(* Logix 5000 project; controller cal1615 1756-L62 rev 20.19; software revision 20.05; part 14 of 81 *)
(* tags used below, declared in another part *)
   FAULT : BOOL;   // Fault AFI
   HMI : BOOL;   // AFI HMI
   p00_lin_timer_pre_0ms : DINT;
   p00_lin_timer_pre_1s : DINT;
   p00_lin_timer_pre_disc : DINT;
   p00_lin_timer_pre_mcp : DINT;
   p00_lin_timer_pre_ms : DINT;
   p00_lin_timer_pre_ol : DINT;
   p01_dint_to_hmi : DINT[16];   // System Dint to HMI
   p01_recipe_active : recipe;   // Active Recipe
   p01r09_pb_global_reset : BOOL;   // System Modes PB: Global Fault Reset
   p02_dint_from_hmi : hmi_dint;
   p02_dint_to_hmi : hmi_dint;   // MOP HMI Iface Dint to HMI
   p02_recipe_from_hmi : recipe;   // MOP HMI Iface Recipe From HMI
   p02_recipe_to_hmi : recipe;   // MOP HMI Iface To HMI Recipe
   p02r01 : routine;   // MOP HMI Iface Main
   p02r02 : routine;   // MOP HMI Iface Misc Control
   p02r02_timer_fault : TIMER[4];   // MOP HMI Iface Misc Control Fault Delay
   p02r02_timer_logout : TIMER;
   p02r02_timer_warning : TIMER[4];   // MOP HMI Iface Misc Control Warning Delay
   p02r03 : routine;   // MOP HMI Iface Navigation
   p02r03_timer_fault : TIMER[4];   // MOP HMI Iface Navigation Fault Delay
   p02r03_timer_warning : TIMER[4];   // MOP HMI Iface Navigation Warning Delay
   p02r04 : routine;   // MOP HMI Iface Recipe
   p02r04_timer_fault : TIMER[4];   // MOP HMI Iface Recipe Fault Delay
   p02r04_timer_warning : TIMER[4];   // MOP HMI Iface Recipe Warning Delay
   p02r05 : routine;   // MOP HMI Iface Dint to HMI
   p02r05_timer_fault : TIMER[4];   // MOP HMI Iface Dint to HMI Fault Delay
   p02r05_timer_warning : TIMER[4];   // MOP HMI Iface Dint to HMI Warning Delay
   p02r07 : routine;   // MOP HMI Iface Alarms
   p11_dint_to_hmi : DINT[16];   // Zone 1 Temperature Control VFDs On
   p12_dint_to_hmi : DINT[16];   // Zone 2 Temperature Control VFDs On
   p13_dint_to_hmi : DINT[16];   // Zone 3 Temperature Control VFDs On
   p19_dint_to_hmi : DINT[16];
   p20_dint_to_hmi : DINT[16];   // Letoff Dint to HMI
   p21_dint_to_hmi : DINT[16];   // Splice Press
   p22_dint_to_hmi : DINT[16];   // Tension Stand 1 Dint to HMI
   p23_dint_to_hmi : DINT[17];   // Impreg Dint to HMI
   p24_dint_to_hmi : DINT[16];
   p25_dint_to_hmi : DINT[16];   // Tension Stand 2 Dint to HMI
   p26_dint_to_hmi : DINT[16];   // Upper Poly Letoff Dint to HMI
   p27_dint_to_hmi : DINT[16];   // Lower Poly Letoff Alarms
   p28_dint_to_hmi : DINT[16];
   p29_dint_to_hmi : DINT[16];   // Winder Dint to HMI
   p30_dint_to_hmi : DINT[16];   // Retraction System Dint to HMI
(* P01_System, continued *)

ROUTINE R32_LIN_Timer_Presets   (* ladder *)
// System
// System Timer Presets
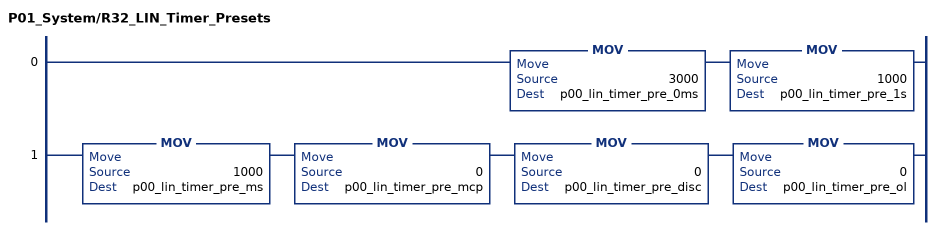
   0: MOV(3000,p00_lin_timer_pre_0ms)MOV(1000,p00_lin_timer_pre_1s);
   1: MOV(1000,p00_lin_timer_pre_ms)MOV(0,p00_lin_timer_pre_mcp)MOV(0,p00_lin_timer_pre_disc)MOV(0,p00_lin_timer_pre_ol);
END_ROUTINE
END_PROGRAM

PROGRAM P02_MOP_HMI_Iface   (* main routine R01_Main *)
VAR
   Limit_Clamp : sys_Limit_Clamp;   // Limit Clamp
END_VAR

ROUTINE R01_Main   (* ladder *)
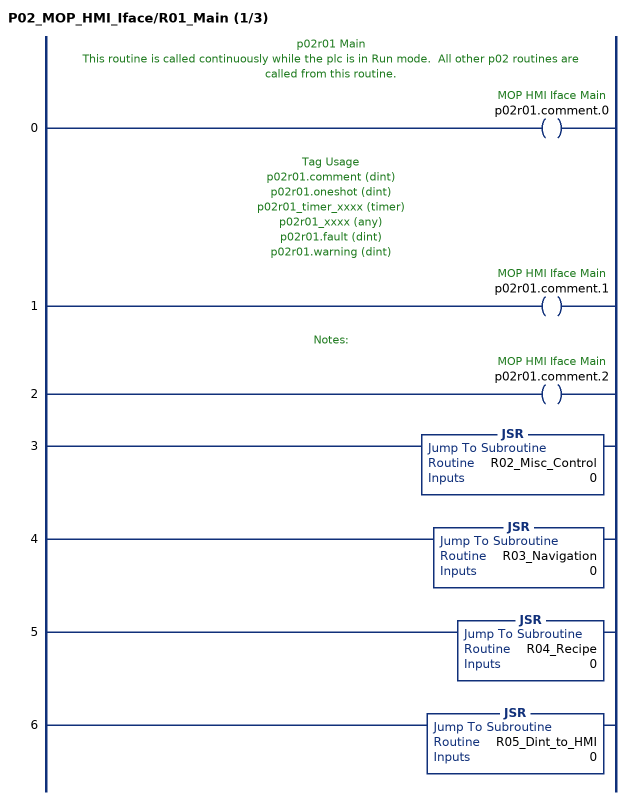
   // p02r01 Main
   // This routine is called continuously while the plc is in Run mode.  All other p02 routines are called from this routine.
   0: OTE(p02r01.comment.0);
   // Tag Usage
   // p02r01.comment (dint)
   // p02r01.oneshot (dint)
   // p02r01_timer_xxxx (timer)
   // p02r01_xxxx (any)
   // p02r01.fault (dint)
   // p02r01.warning (dint)
   1: OTE(p02r01.comment.1);
   // Notes:
   2: OTE(p02r01.comment.2);
   3: JSR(R02_Misc_Control,0);
   4: JSR(R03_Navigation,0);
   5: JSR(R04_Recipe,0);
   6: JSR(R05_Dint_to_HMI,0);
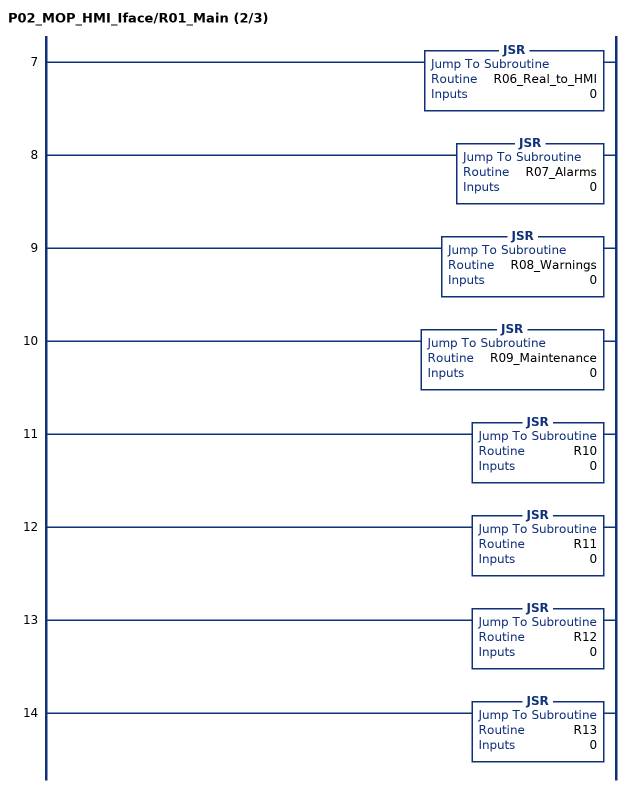
   7: JSR(R06_Real_to_HMI,0);
   8: JSR(R07_Alarms,0);
   9: JSR(R08_Warnings,0);
   10: JSR(R09_Maintenance,0);
   11: JSR(R10,0);
   12: JSR(R11,0);
   13: JSR(R12,0);
   14: JSR(R13,0);
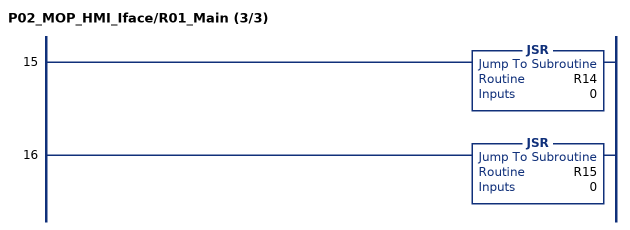
   15: JSR(R14,0);
   16: JSR(R15,0);
END_ROUTINE

ROUTINE R02_Misc_Control   (* ladder *)
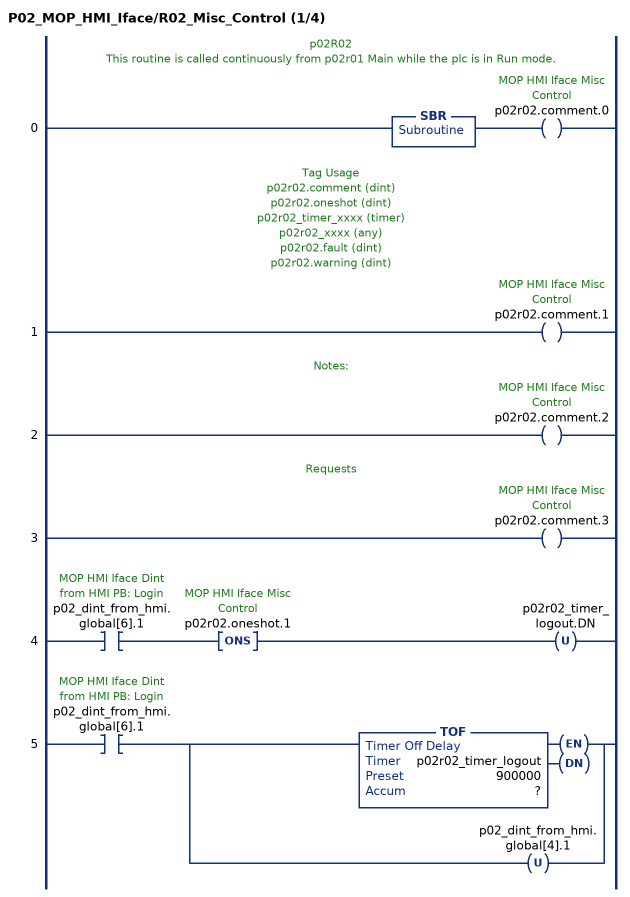
   // p02R02
   // This routine is called continuously from p02r01 Main while the plc is in Run mode.
   0: SBR()OTE(p02r02.comment.0);
   // Tag Usage
   // p02r02.comment (dint)
   // p02r02.oneshot (dint)
   // p02r02_timer_xxxx (timer)
   // p02r02_xxxx (any)
   // p02r02.fault (dint)
   // p02r02.warning (dint)
   1: OTE(p02r02.comment.1);
   // Notes:
   2: OTE(p02r02.comment.2);
   // Requests
   3: OTE(p02r02.comment.3);
   4: XIC(p02_dint_from_hmi.global[6].1)ONS(p02r02.oneshot.1)OTU(p02r02_timer_logout.DN);
   5: XIC(p02_dint_from_hmi.global[6].1)[TOF(p02r02_timer_logout,?,?) ,OTU(p02_dint_from_hmi.global[4].1) ];
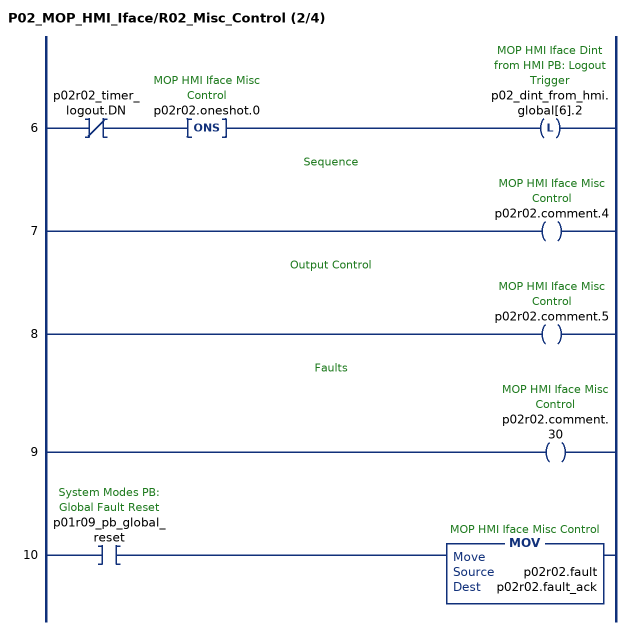
   6: XIO(p02r02_timer_logout.DN)ONS(p02r02.oneshot.0)OTL(p02_dint_from_hmi.global[6].2);
   // Sequence
   7: OTE(p02r02.comment.4);
   // Output Control
   8: OTE(p02r02.comment.5);
   // Faults
   9: OTE(p02r02.comment.30);
   10: XIC(p01r09_pb_global_reset)MOV(p02r02.fault,p02r02.fault_ack);
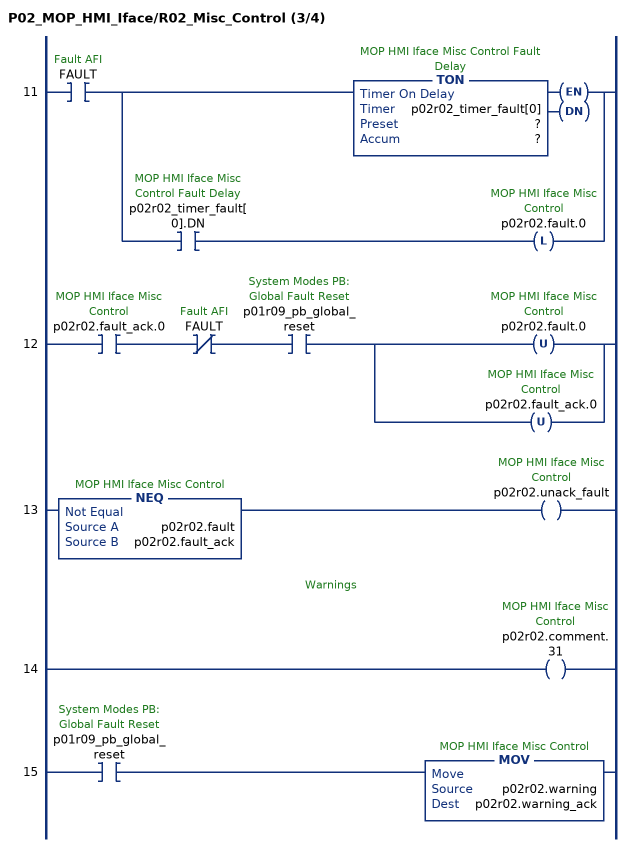
   11: XIC(FAULT)[TON(p02r02_timer_fault[0],?,?) ,XIC(p02r02_timer_fault[0].DN) OTL(p02r02.fault.0) ];
   12: XIC(p02r02.fault_ack.0)XIO(FAULT)XIC(p01r09_pb_global_reset)[OTU(p02r02.fault.0) ,OTU(p02r02.fault_ack.0) ];
   13: NEQ(p02r02.fault,p02r02.fault_ack)OTE(p02r02.unack_fault);
   // Warnings
   14: OTE(p02r02.comment.31);
   15: XIC(p01r09_pb_global_reset)MOV(p02r02.warning,p02r02.warning_ack);
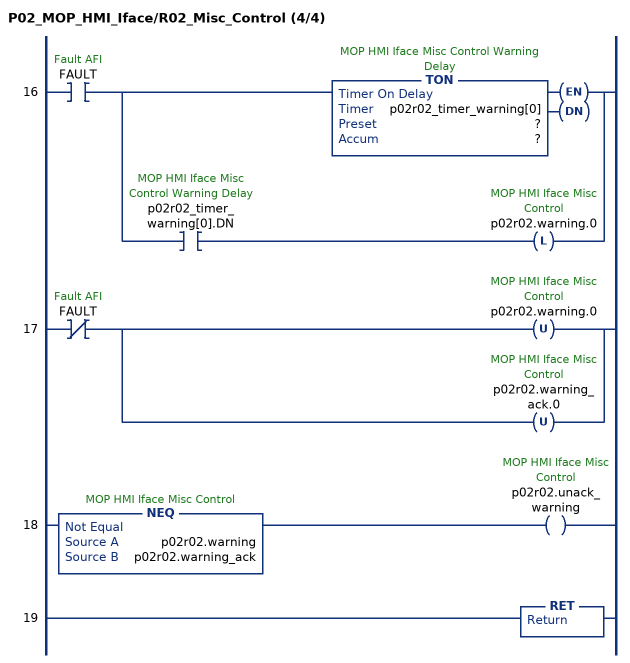
   16: XIC(FAULT)[TON(p02r02_timer_warning[0],?,?) ,XIC(p02r02_timer_warning[0].DN) OTL(p02r02.warning.0) ];
   17: XIO(FAULT)[OTU(p02r02.warning.0) ,OTU(p02r02.warning_ack.0) ];
   18: NEQ(p02r02.warning,p02r02.warning_ack)OTE(p02r02.unack_warning);
   19: RET();
END_ROUTINE

ROUTINE R03_Navigation   (* ladder *)
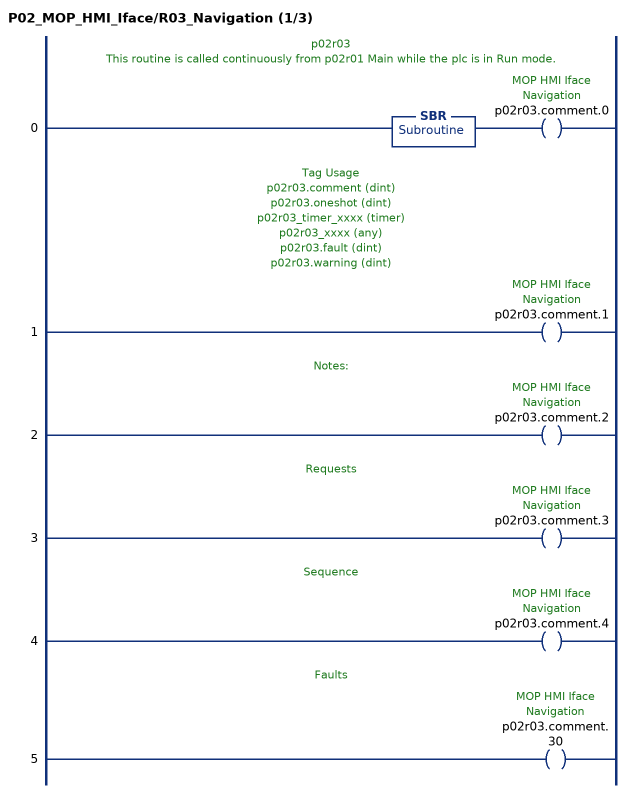
   // p02r03
   // This routine is called continuously from p02r01 Main while the plc is in Run mode.
   0: SBR()OTE(p02r03.comment.0);
   // Tag Usage
   // p02r03.comment (dint)
   // p02r03.oneshot (dint)
   // p02r03_timer_xxxx (timer)
   // p02r03_xxxx (any)
   // p02r03.fault (dint)
   // p02r03.warning (dint)
   1: OTE(p02r03.comment.1);
   // Notes:
   2: OTE(p02r03.comment.2);
   // Requests
   3: OTE(p02r03.comment.3);
   // Sequence
   4: OTE(p02r03.comment.4);
   // Faults
   5: OTE(p02r03.comment.30);
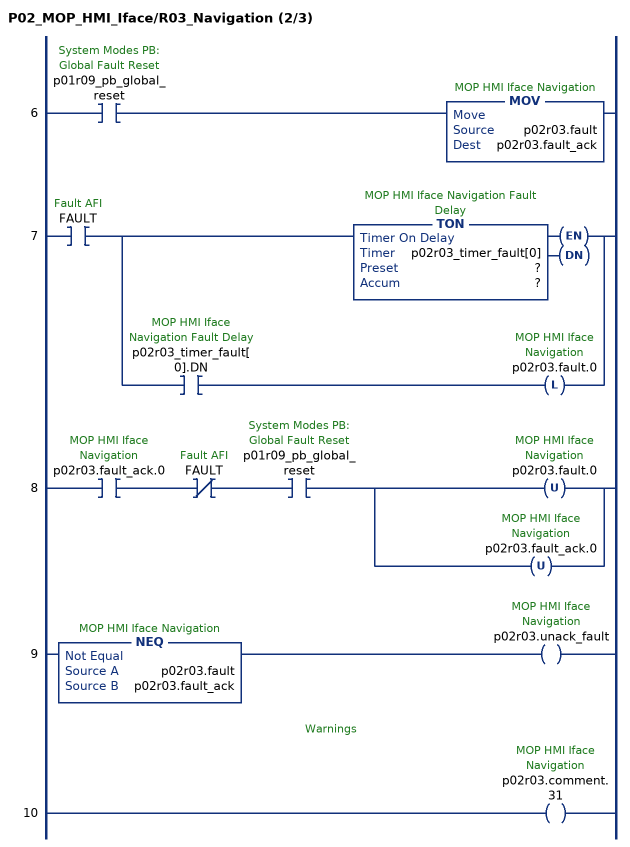
   6: XIC(p01r09_pb_global_reset)MOV(p02r03.fault,p02r03.fault_ack);
   7: XIC(FAULT)[TON(p02r03_timer_fault[0],?,?) ,XIC(p02r03_timer_fault[0].DN) OTL(p02r03.fault.0) ];
   8: XIC(p02r03.fault_ack.0)XIO(FAULT)XIC(p01r09_pb_global_reset)[OTU(p02r03.fault.0) ,OTU(p02r03.fault_ack.0) ];
   9: NEQ(p02r03.fault,p02r03.fault_ack)OTE(p02r03.unack_fault);
   // Warnings
   10: OTE(p02r03.comment.31);
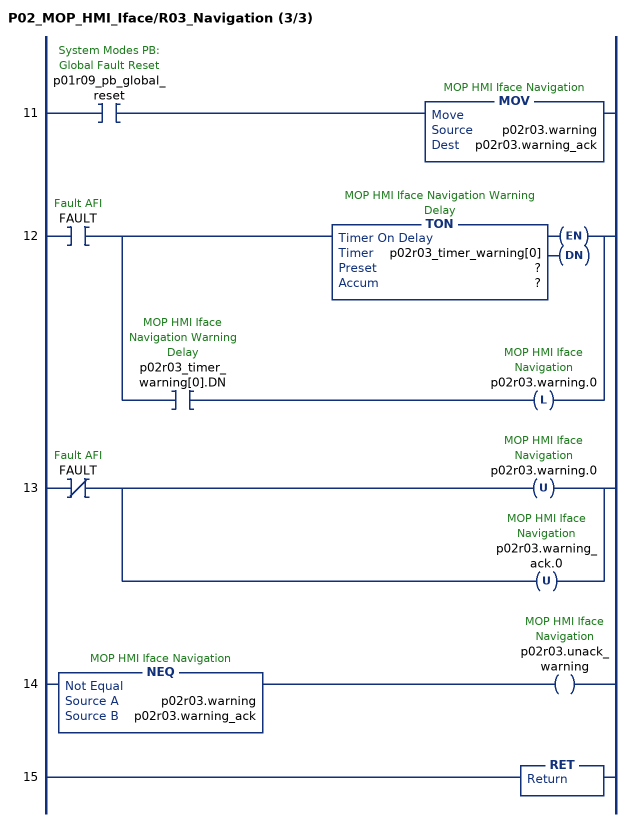
   11: XIC(p01r09_pb_global_reset)MOV(p02r03.warning,p02r03.warning_ack);
   12: XIC(FAULT)[TON(p02r03_timer_warning[0],?,?) ,XIC(p02r03_timer_warning[0].DN) OTL(p02r03.warning.0) ];
   13: XIO(FAULT)[OTU(p02r03.warning.0) ,OTU(p02r03.warning_ack.0) ];
   14: NEQ(p02r03.warning,p02r03.warning_ack)OTE(p02r03.unack_warning);
   15: RET();
END_ROUTINE

ROUTINE R04_Recipe   (* ladder *)
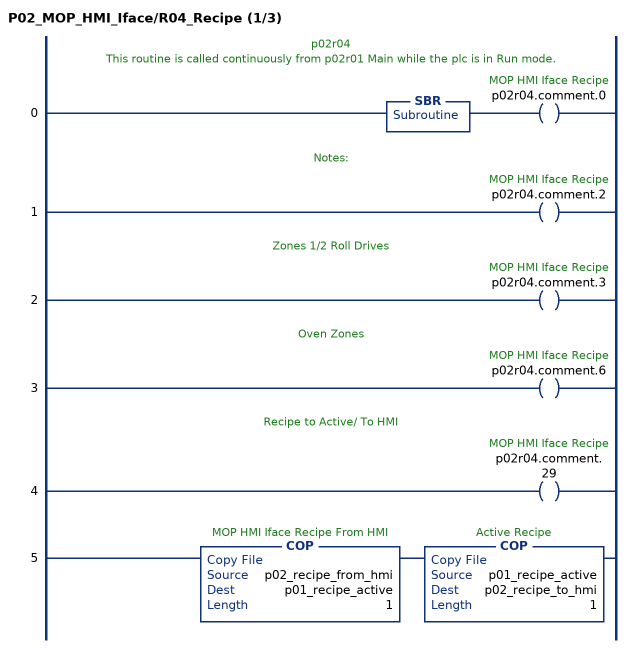
   // p02r04
   // This routine is called continuously from p02r01 Main while the plc is in Run mode.
   0: SBR()OTE(p02r04.comment.0);
   // Notes:
   1: OTE(p02r04.comment.2);
   // Zones 1/2 Roll Drives
   2: OTE(p02r04.comment.3);
   // Oven Zones
   3: OTE(p02r04.comment.6);
   // Recipe to Active/ To HMI
   4: OTE(p02r04.comment.29);
   5: COP(p02_recipe_from_hmi,p01_recipe_active,1)COP(p01_recipe_active,p02_recipe_to_hmi,1);
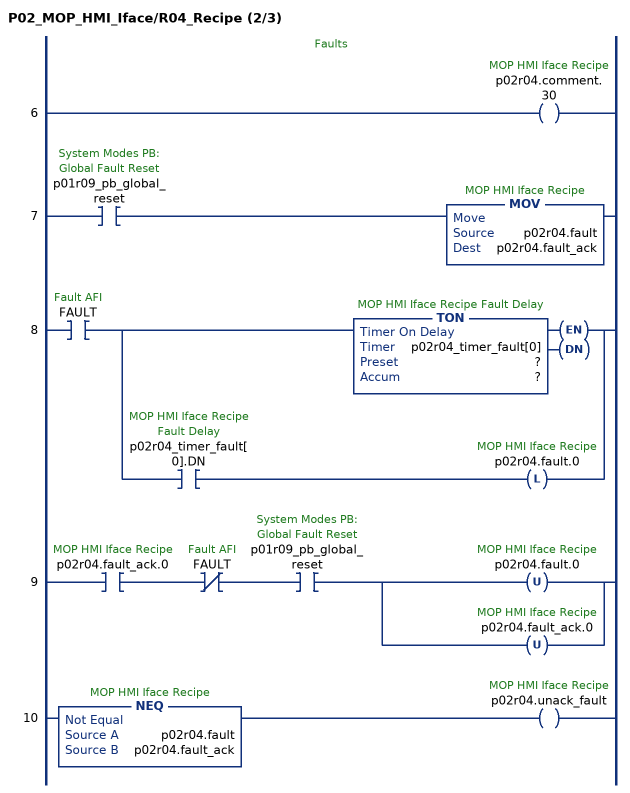
   // Faults
   6: OTE(p02r04.comment.30);
   7: XIC(p01r09_pb_global_reset)MOV(p02r04.fault,p02r04.fault_ack);
   8: XIC(FAULT)[TON(p02r04_timer_fault[0],?,?) ,XIC(p02r04_timer_fault[0].DN) OTL(p02r04.fault.0) ];
   9: XIC(p02r04.fault_ack.0)XIO(FAULT)XIC(p01r09_pb_global_reset)[OTU(p02r04.fault.0) ,OTU(p02r04.fault_ack.0) ];
   10: NEQ(p02r04.fault,p02r04.fault_ack)OTE(p02r04.unack_fault);
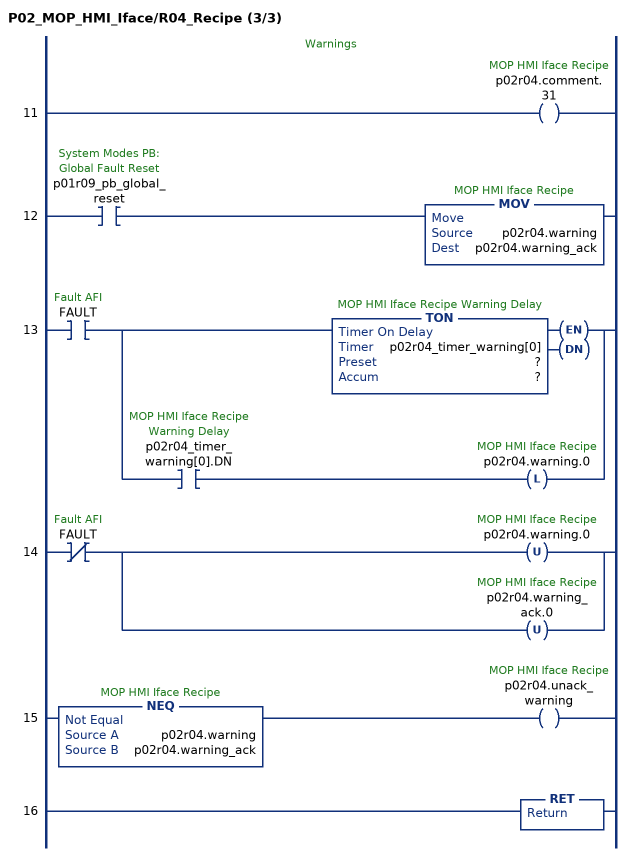
   // Warnings
   11: OTE(p02r04.comment.31);
   12: XIC(p01r09_pb_global_reset)MOV(p02r04.warning,p02r04.warning_ack);
   13: XIC(FAULT)[TON(p02r04_timer_warning[0],?,?) ,XIC(p02r04_timer_warning[0].DN) OTL(p02r04.warning.0) ];
   14: XIO(FAULT)[OTU(p02r04.warning.0) ,OTU(p02r04.warning_ack.0) ];
   15: NEQ(p02r04.warning,p02r04.warning_ack)OTE(p02r04.unack_warning);
   16: RET();
END_ROUTINE

ROUTINE R05_Dint_to_HMI   (* ladder *)
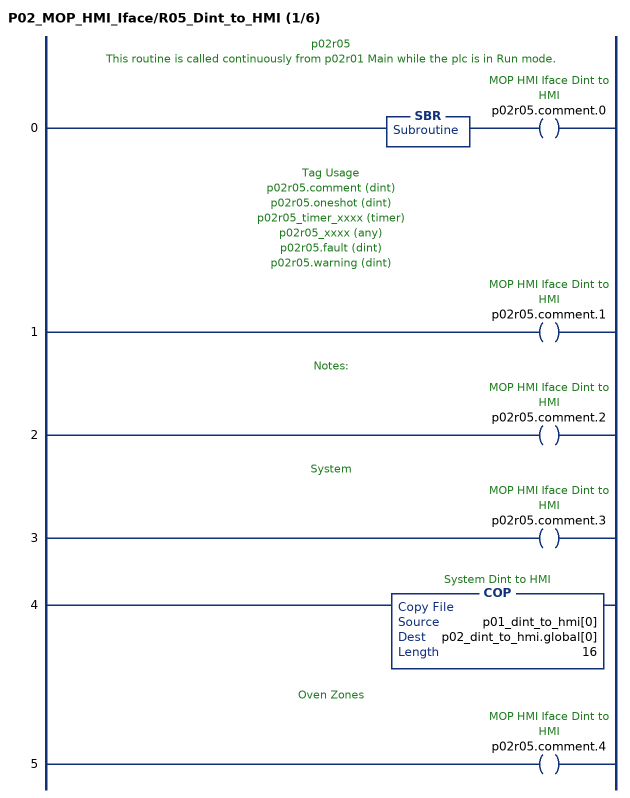
   // p02r05
   // This routine is called continuously from p02r01 Main while the plc is in Run mode.
   0: SBR()OTE(p02r05.comment.0);
   // Tag Usage
   // p02r05.comment (dint)
   // p02r05.oneshot (dint)
   // p02r05_timer_xxxx (timer)
   // p02r05_xxxx (any)
   // p02r05.fault (dint)
   // p02r05.warning (dint)
   1: OTE(p02r05.comment.1);
   // Notes:
   2: OTE(p02r05.comment.2);
   // System
   3: OTE(p02r05.comment.3);
   4: COP(p01_dint_to_hmi[0],p02_dint_to_hmi.global[0],16);
   // Oven Zones
   5: OTE(p02r05.comment.4);
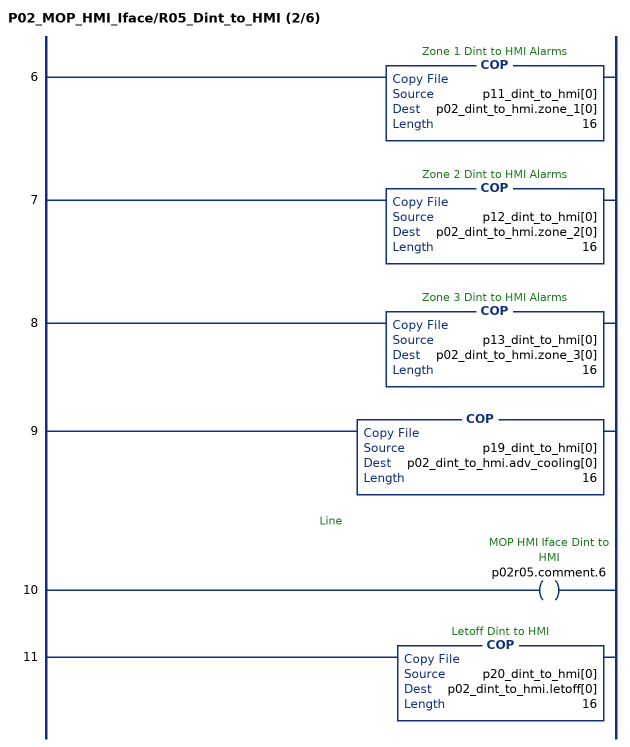
   6: COP(p11_dint_to_hmi[0],p02_dint_to_hmi.zone_1[0],16);
   7: COP(p12_dint_to_hmi[0],p02_dint_to_hmi.zone_2[0],16);
   8: COP(p13_dint_to_hmi[0],p02_dint_to_hmi.zone_3[0],16);
   9: COP(p19_dint_to_hmi[0],p02_dint_to_hmi.adv_cooling[0],16);
   // Line
   10: OTE(p02r05.comment.6);
   11: COP(p20_dint_to_hmi[0],p02_dint_to_hmi.letoff[0],16);
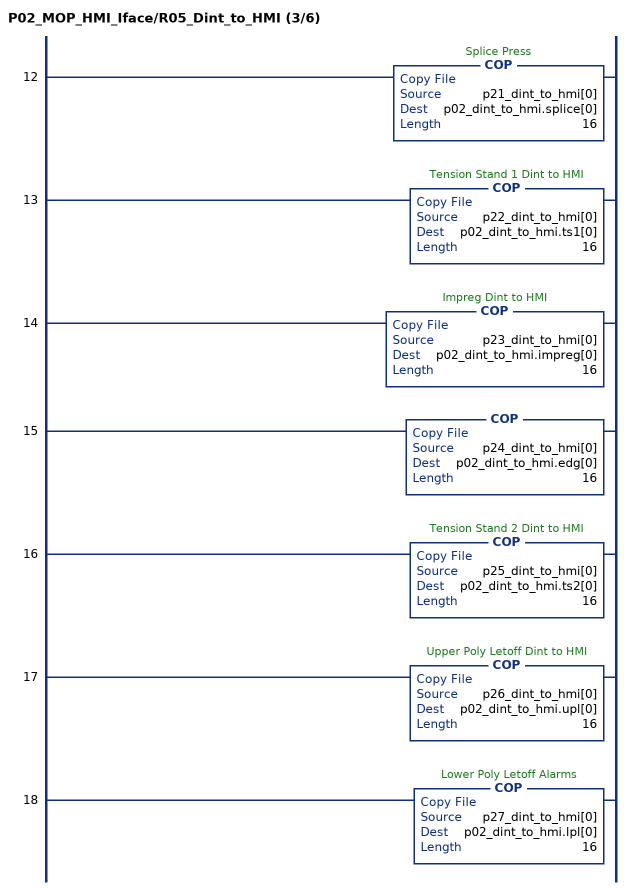
   12: COP(p21_dint_to_hmi[0],p02_dint_to_hmi.splice[0],16);
   13: COP(p22_dint_to_hmi[0],p02_dint_to_hmi.ts1[0],16);
   14: COP(p23_dint_to_hmi[0],p02_dint_to_hmi.impreg[0],16);
   15: COP(p24_dint_to_hmi[0],p02_dint_to_hmi.edg[0],16);
   16: COP(p25_dint_to_hmi[0],p02_dint_to_hmi.ts2[0],16);
   17: COP(p26_dint_to_hmi[0],p02_dint_to_hmi.upl[0],16);
   18: COP(p27_dint_to_hmi[0],p02_dint_to_hmi.lpl[0],16);
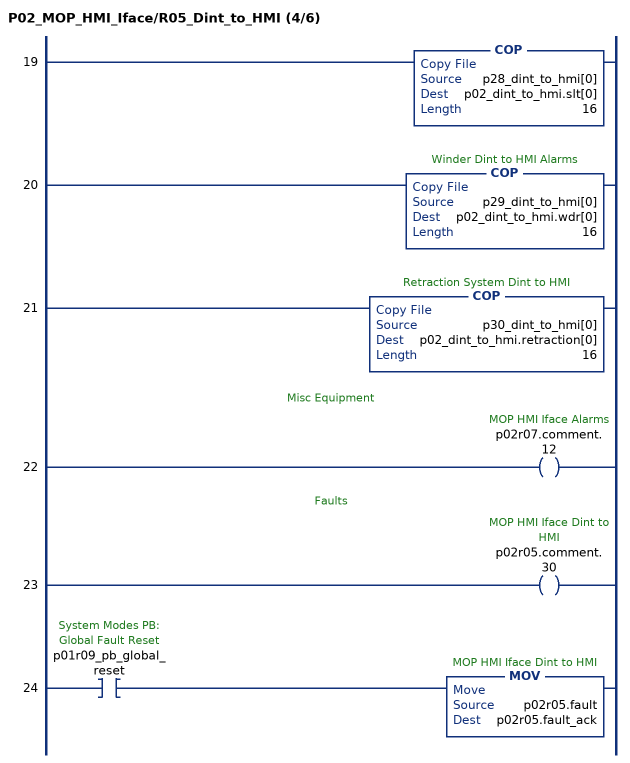
   19: COP(p28_dint_to_hmi[0],p02_dint_to_hmi.slt[0],16);
   20: COP(p29_dint_to_hmi[0],p02_dint_to_hmi.wdr[0],16);
   21: COP(p30_dint_to_hmi[0],p02_dint_to_hmi.retraction[0],16);
   // Misc Equipment
   22: OTE(p02r07.comment.12);
   // Faults
   23: OTE(p02r05.comment.30);
   24: XIC(p01r09_pb_global_reset)MOV(p02r05.fault,p02r05.fault_ack);
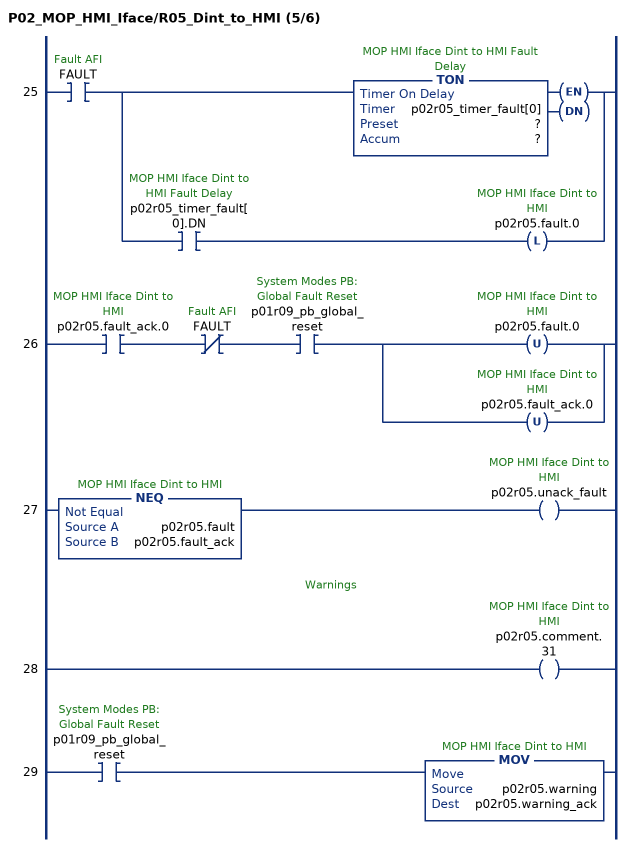
   25: XIC(FAULT)[TON(p02r05_timer_fault[0],?,?) ,XIC(p02r05_timer_fault[0].DN) OTL(p02r05.fault.0) ];
   26: XIC(p02r05.fault_ack.0)XIO(FAULT)XIC(p01r09_pb_global_reset)[OTU(p02r05.fault.0) ,OTU(p02r05.fault_ack.0) ];
   27: NEQ(p02r05.fault,p02r05.fault_ack)OTE(p02r05.unack_fault);
   // Warnings
   28: OTE(p02r05.comment.31);
   29: XIC(p01r09_pb_global_reset)MOV(p02r05.warning,p02r05.warning_ack);
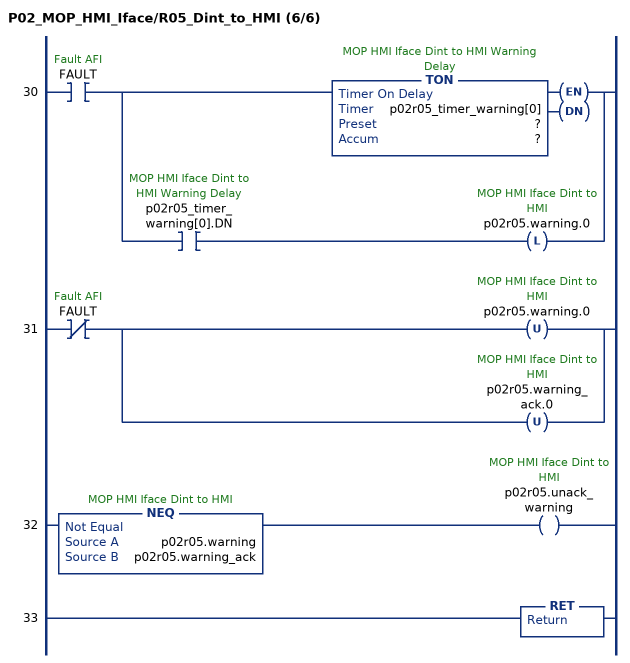
   30: XIC(FAULT)[TON(p02r05_timer_warning[0],?,?) ,XIC(p02r05_timer_warning[0].DN) OTL(p02r05.warning.0) ];
   31: XIO(FAULT)[OTU(p02r05.warning.0) ,OTU(p02r05.warning_ack.0) ];
   32: NEQ(p02r05.warning,p02r05.warning_ack)OTE(p02r05.unack_warning);
   33: RET();
END_ROUTINE
